PROGRAM MAIN
VAR
//	{attribute 'TcLinkTo' := '.bLimFwd:=TIIB[y_up]^STM Status^Status^Digital input 1; .bLimBwd:=TIIB[y_up]^STM Status^Status^Digital input 2; .bSTO:=TIIB[di]^Channel 1^Input'}	
	{attribute 'TcLinkTo':='.bLimFwd:=TIIB[y_up]^STM Status^Status^Digital input 1'}		
    M1: DUT_MotionStage:=(nCommand:=3); // Yup
//	{attribute 'TcLinkTo' := '.bLimFwd:=TIIB[y_dwn]^STM Status^Status^Digital input 1; .bLimBwd:=TIIB[y_dwn]^STM Status^Status^Digital input 2'}
	M2: DUT_MotionStage:=(nCommand:=3); // Ydwn
//	{attribute 'TcLinkTo' := '.bLimFwd:=TIIB[x_up]^STM Status^Status^Digital input 1; .bLimBwd:=TIIB[x_up]^STM Status^Status^Digital input 2'}	
	M3: DUT_MotionStage:=(nCommand:=3); // Xup
//	{attribute 'TcLinkTo' := '.bLimFwd:=TIIB[x_dwn]^STM Status^Status^Digital input 1; .bLimBwd:=TIIB[x_dwn]^STM Status^Status^Digital input 2'}
	M4: DUT_MotionStage:=(nCommand:=3); // Xdwn
//	{attribute 'TcLinkTo' := '.bLimFwd:=TIIB[pitch]^STM Status^Status^Digital input 1; .bLimBwd:=TIIB[pitch]^STM Status^Status^Digital input 2'}	
	M5: DUT_MotionStage:=(nCommand:=3); // PitchCoarse
	fbMotionStage_x_up, fbMotionStage_x_dwn, fbMotionStage_y_up, fbMotionStage_y_dwn, fbMotionStage_pitch : FB_MotionStage;
	stoEnable AT %I* : BOOL;
	{attribute 'TcLinkTo' := '.Count:=TIIB[1-x_up_2-x_dwn]^FB Inputs Channel 1^Position'}	
	x_up_enc  AT %I*: ST_RenishawAbsEnc;
	{attribute 'TcLinkTo' := '.Count:=TIIB[1-x_up_2-x_dwn]^FB Inputs Channel 2^Position'}
	x_dwn_enc  AT %I*: ST_RenishawAbsEnc;
	{attribute 'TcLinkTo' := '.Count:=TIIB[1-y_up_2-y_dwn]^FB Inputs Channel 1^Position'}	
	y_up_enc  AT %I*: ST_RenishawAbsEnc;
	{attribute 'TcLinkTo' := '.Count:=TIIB[1-y_up_2-y_dwn]^FB Inputs Channel 2^Position'}
	y_dwn_enc  AT %I*: ST_RenishawAbsEnc;
	// Auto coupling function block
	fbAutoCoupleX : FB_GantryAutoCoupling;
	fbAutoCoupleY : FB_GantryAutoCoupling;
	bExecuteCoupleX : BOOL;
	bExecuteCoupleY : BOOL;
	bExecuteDecoupleX : BOOL;
	bExecuteDecoupleY : BOOL;
	bGantryAlreadyCoupledX : BOOL;
	bGantryAlreadyCoupledY : BOOL;
	
	// Gantry variables
	nCurrGantryX : LINT;
	nCurrGantryY : LINT;
	nGantryTolX : LINT := 25000;
	nGantryTolY : LINT := 25000;
END_VAR

// M1K2
// Buttons to enable motors: write 0 to enable, 2 to disable
M1.nEnableMode; // Yup
M2.nEnableMode; // Ydwn
M3.nEnableMode; // Xup
M4.nEnableMode; // Xdwn
M5.nEnableMode; // PitchCoarse

// Encoder Reference Values: Taking from Axilon FAT
//M1K2 Ref Vals
y_up_enc.Ref := 64970000;
y_dwn_enc.Ref := 65030000; // Use initial motor positions for now
x_up_enc.Ref := 20302000;
x_dwn_enc.Ref := 21280500;

// Gantry Differences to monitor
nCurrGantryY := ((ULINT_TO_LINT(y_up_enc.Count) - ULINT_TO_LINT(y_up_enc.Ref)) - (ULINT_TO_LINT(y_dwn_enc.Count) - ULINT_TO_LINT(y_dwn_enc.Ref)));
nCurrGantryX := ((ULINT_TO_LINT(x_up_enc.Count) - ULINT_TO_LINT(x_up_enc.Ref)) - (ULINT_TO_LINT(x_dwn_enc.Count) - ULINT_TO_LINT(x_dwn_enc.Ref)));

// E-stop
M1.bHardwareEnable := stoEnable;
M2.bHardwareEnable := stoEnable;
M3.bHardwareEnable := stoEnable;
M4.bHardwareEnable := stoEnable;
M5.bHardwareEnable := stoEnable;


// Start Autocoupling
fbAutoCoupleX(nGantryTol:=nGantryTolX, Master:=M3, MasterEnc:=x_up_enc, Slave:=M4,
	          SlaveEnc:=x_dwn_enc, bExecuteCouple:=bExecuteCoupleX,
              bExecuteDecouple:=bExecuteDecoupleX,
              bGantryAlreadyCoupled=>bGantryAlreadyCoupledX);

fbAutoCoupleY(nGantryTol:=nGantryTolY, Master:=M1, MasterEnc:=y_up_enc, Slave:=M2,
	          SlaveEnc:=y_dwn_enc, bExecuteCouple:=bExecuteCoupleY,
              bExecuteDecouple:=bExecuteDecoupleY,
			  bGantryAlreadyCoupled=>bGantryAlreadyCoupledY);

fbMotionStage_y_up  (stMotionStage:=M1);
fbMotionStage_y_dwn (stMotionStage:=M2);
fbMotionStage_x_up  (stMotionStage:=M3);
fbMotionStage_x_dwn (stMotionStage:=M4);
fbMotionStage_pitch (stMotionStage:=M5);

END_PROGRAM

(* stored: Version 1.1.0.1, ProductVersion 3.1.4022.18
   POU MAIN: Id {2ce36a91-321d-4828-96a2-d7e21b9a58d0}, SpecialFunc None *)
